(* Logix 5000 project; controller BigNumber Emulate 5570 rev 30.12; software revision 30.00 *)

TASK MainTask (periodic, rate 12000 ms, priority 1, watchdog 12000 ms) : MainProgram

MODULES
   Local : Emulate 5570 (ICP 3, rev 30.12)
       : vendor 1 type 0 code 15 (ICP 0, rev 1.1, Output RPI 50 ms)
END_MODULES

VAR_GLOBAL   (* controller tags *)
   SCAN_CYCLE_TIME : DINT; {access None}
END_VAR

PROGRAM MainProgram   (* main routine MainRoutine *)
VAR
   Add_c : DINT; {access None}
   Add_Digits : DINT; {access None}
   Add_i : DINT; {access None}
   Add_input_x : DINT[512]; {access None}
   Add_input_y : DINT[512]; {access None}
   Add_j : DINT; {access None}
   Add_Result : DINT[513]; {access None}
   Add_tmp : DINT;
   AddMul_2Base : DINT[250];
   AddMul_Base : DINT[249];
   AddMul_Digits : DINT;
   AddMul_exp_bitindx : DINT;
   AddMul_exp_blk : DINT;
   AddMul_i : DINT;
   AddMul_input_exp : DINT[249];
   AddMul_input_g : DINT[249];
   AddMul_j : DINT;
   AddMul_Result : DINT[500];
   Big_base : DINT; {access None}
   Big_Comp_i : DINT;
   Big_Comp_Res : DINT;
   Big_lb : DINT;
   Big_Ver : DINT;
   Div_Digits : DINT; {access None}
   Div_i : DINT; {access None}
   Div_input_x : DINT[500]; {access None}
   Div_input_y : DINT[500]; {access None}
   Div_j : DINT; {access None}
   Div_k : DINT; {access None}
   Div_m : DINT; {access None}
   Div_mul : DINT[500]; {access None}
   Div_q_Digits : DINT; {access None}
   Div_quotient : DINT[500]; {access None}
   Div_remainder : DINT[500]; {access None}
   Div_state : DINT; {access None}
   Div_sub_n : DINT; {access None}
   Div_x : DINT; {access None}
   Div_x_Digits : DINT; {access None}
   Div_y_Digits : DINT; {access None}
   Mul_c : DINT; {access None}
   Mul_Comp : DINT; {access None}
   Mul_Digits : DINT; {access None}
   Mul_i : DINT; {access None}
   Mul_input_x : DINT[513]; {access None}
   Mul_input_y : DINT[513]; {access None}
   Mul_j : DINT; {access None}
   Mul_q : DINT; {access None}
   Mul_Result : DINT[1025]; {access None}
   Mul_u : DINT; {access None}
   Mul_v : DINT; {access None}
   Mul_x : DINT; {access None}
   Mul_y : DINT; {access None}
   Sub_c : DINT; {access None}
   Sub_Digits : DINT; {access None}
   Sub_i : DINT; {access None}
   Sub_input_x : DINT[512]; {access None}
   Sub_input_y : DINT[512]; {access None}
   Sub_j : DINT; {access None}
   Sub_Result : DINT[512]; {access None}
END_VAR

ROUTINE BIGINTEGER_Add   (* structured text *)
   //Calculate the addition of big numbers.  Resource: page 594 of the handbook.
   //input positive big intergers  Add_input_x[] and Add_input_y[], each having UHF_sints base UHF_base digits.
   //output: the sum Add_Result[] in radix UHF_base representation.
   
   // Addition test
   (*if S:FS then
   	Add_Digits:= 10;  //the Digits of input.
   	UHF_base:= 10; //input in decimal
   	// Addition test
   	for Add_i:=0 to Add_Digits-1 by 1 do //assign value to input
   		Add_input_x[Add_i]:=9;
   		Add_input_y[Add_i]:=9;
   	end_for;
   end_if; *)
   
   //JSR(BIGINTEGER_Init);
   
   
   
   for Add_i:=0 to Add_Digits by 1 do
   	Add_Result[Add_i]:=0;  //Initialize the sum to 0.
   end_for;
   
   //Calculate the sum Add_input_x[] + Add_input_y[].
   Add_c.[0]:=0;   //Initialize carry to zero.
   
   for Add_j:=0 to Add_Digits-1 by 1 do
   	Add_Result[Add_j]:=Add_input_x[Add_j] + Add_input_y[Add_j] + Add_c; // Compute every digit of the sum.
   
   	Case Big_Ver OF
   	0:
   		if Add_Result[Add_j]> Big_base Then
   			Add_c:=1;
   		else
   			Add_c:=0;
   		End_if;
   		Add_Result[Add_j]:= Add_tmp mod Big_base;
   	1,2:
   		Add_c.[0]:=Add_Result[Add_j].[Big_lb];
   		Add_Result[Add_j].[Big_lb]:=0;	//最高位清零
   	End_Case;
   end_for;
   
   Add_Result[Add_Digits]:= Add_c;
   
   Add_c:=0;
   
END_ROUTINE

ROUTINE BIGINTEGER_AMul   (* structured text *)
   //Input: g ∈ G, whereGisanadditivegroup,andapositiveintegere = (e_t, e_t−1 ···e _1 e_ 0 ) 2 .
   //OUTPUT: e · g.
   
   
   //A←0.
   //2. For i from t down to 0 do the following:
   //2.1 A←A + A.
   //2.2 If e i = 1 then A←A + g.
   //3. Return(A).
   
   /////////////////////////////////////////////////////////////////////////////////////////////
   
   
   For AddMul_i:=0 to AddMul_Digits-1 by 1 Do
   	AddMul_Result[AddMul_i]:=0;
   End_For;
   AddMul_exp_bitindx:=29; //indexing 30bits
   AddMul_exp_blk:=AddMul_Digits-2;
   
   
   For AddMul_i:=AddMul_Digits-2 to 0 by -1 Do
   	While AddMul_exp_bitindx>=0 Do
   		if AddMul_i<> AddMul_Digits-2 or AddMul_exp_bitindx <> 29 Then
   			Add_Digits:= AddMul_Digits-1;
   				for Add_i:=0 to Add_Digits-1 by 1 do //assign value to input
   					Add_input_x[Add_i]:=AddMul_Result[Add_i];
   					Add_input_y[Add_i]:=AddMul_Result[Add_i];
   				end_for;
   			JSR(BIGINTEGER_Add);
   			for Add_i:=0 to Add_Digits by 1 do //
   				AddMul_Result[Add_i]:=Add_Result[Add_i];
   			end_for;
   
   			JSR(BIGINTEGER_Comparison);
   			If Big_Comp_Res=1 Then           //mod m
   				Sub_Digits:= AddMul_Digits-1;
   				for Sub_i:=0 to Sub_Digits-1 by 1 do //assign value to input
   					Add_input_x[Sub_i]:=AddMul_Result[Sub_i];
   					Add_input_y[Sub_i]:=AddMul_Base[Sub_i];
   				end_for;
   				JSR(BIGINTEGER_Sub);
   				for Sub_i:=0 to Add_Digits by 1 do //
   					AddMul_Result[Sub_i]:=Add_Result[Sub_i];
   				end_for;
   			End_If;
   
   		End_IF;
   
   
   
   		If AddMul_input_exp[AddMul_exp_blk].[AddMul_exp_bitindx] Then
   			Add_Digits:= AddMul_Digits-1;
   				for Add_i:=0 to Add_Digits-1 by 1 do //assign value to input
   					Add_input_x[Add_i]:=AddMul_Result[Add_i];
   					Add_input_y[Add_i]:=AddMul_input_g[Add_i];
   				end_for;
   			JSR(BIGINTEGER_Add);
   			for Add_i:=0 to Add_Digits by 1 do //
   				AddMul_Result[Add_i]:=Add_Result[Add_i];
   			end_for;
   
   			JSR(BIGINTEGER_Comparison);
   			If Big_Comp_Res=1 Then           //mod m
   				Sub_Digits:= AddMul_Digits-1;
   				for Sub_i:=0 to Sub_Digits-1 by 1 do //assign value to input
   					Add_input_x[Sub_i]:=AddMul_Result[Sub_i];
   					Add_input_y[Sub_i]:=AddMul_Base[Sub_i];
   				end_for;
   				JSR(BIGINTEGER_Sub);
   				for Sub_i:=0 to Add_Digits by 1 do //
   					AddMul_Result[Sub_i]:=Add_Result[Sub_i];
   				end_for;
   			End_If;
   
   		End_If;
   		AddMul_exp_bitindx:=AddMul_exp_bitindx-1;
   
   	End_while;
   
   
   	AddMul_exp_blk:=AddMul_exp_blk-1;
   	AddMul_exp_bitindx:=29;
   
   
   End_For;
   
   
   
   
   
END_ROUTINE

ROUTINE BIGINTEGER_Comparison   (* structured text *)
   Big_Comp_Res:=0;    //0: x>=y,  1: x<y
   
   
   Big_Comp_i:=AddMul_Digits-1;
   
   
   While Big_Comp_i>= 0 do
   
   	if AddMul_2Base[Big_Comp_i]< AddMul_Result[Big_Comp_i] Then
   	 	Big_Comp_Res:=1;
   		exit;
   	End_If;
   
   	Big_Comp_i:=Big_Comp_i-1;
   
   End_while;
   
   
   
END_ROUTINE

ROUTINE BIGINTEGER_Div   (* structured text *)
   //Calculate the division of big numbers.  Resource: page 598 of the handbook.
   //input positive big intergers  Div_input_x[] and Div_input_y[], Div_input_x[] having UHF_sints base UHF_base digits.
   //output: the quotient Div_quo[] and remainder Div_rem[] in radix UHF_base representation.
   
   (*if S:FS then
   	// division test
   	Div_state:=0;
    	Div_Digits:= 10;  //the Digits of input.
   	UHF_base:= 10; //input in decimal
   	for Div_i:=0 to Div_Digits-1 by 1 do   //assign value to input
   		Div_input_x[Div_i]:=9;
   	end_for;
   	for Div_i:=0 to (Div_Digits-1)/2 by 1 do
   		Div_input_y[Div_i]:=9;
   	end_for;
   end_if;*)
   
   	for Div_i:=Div_Digits-1 to 0 by -1 do  //Calculate the numbers of digit of Div_input_x[].
   		if Div_input_x[Div_i] <> 0 then
   			Div_x_Digits:= Div_i;
   			exit;
   		end_if;
   	end_for;
   
   	for Div_i:=Div_Digits-1 to 0 by -1 do  ////Calculate the numbers of digits of Div_input_y[].
   		if Div_input_y[Div_i] <> 0 then
   			Div_y_Digits:= Div_i;
   			exit;
   		end_if;
   	end_for;
   
   	Div_q_Digits:= Div_x_Digits - Div_y_Digits; //the numbers of digit of Div_quotient[].
   	for Div_i:=0 to Div_q_Digits by 1 do
   		Div_quotient[Div_i]:= 0;    //Initialize Div_quotient[] is zero.
   	end_for;
   
   	for Div_i:=0 to Div_x_Digits by 1 do
   		Div_mul[Div_i]:=0;
   	end_for;
   
   
   //When the dividend is less than the divisor, e.g Div_input_x is less than Div_input_y
   for Div_i:=Div_Digits-1 to 0 by -1 do
   	if Div_x_Digits <= Div_y_Digits and Div_input_x[Div_i] < Div_input_y[Div_i] then
   		Div_quotient[0]:=0;
   		for Div_i:=0 to Div_x_Digits by 1 do
   			Div_remainder[Div_i]:=Div_input_x[Div_i];
   		end_for;
   		exit;
   	else
   		Div_state:=1;
   	end_if;
   end_for;
   
   //When the dividend is equal to the divisor
   if Div_state=1 then
   	for Div_i:=Div_Digits-1 to 0 by -1 do
   		if Div_x_Digits = Div_y_Digits and Div_input_x[Div_i] = Div_input_y[Div_i] then
   			Div_quotient[0]:= 1;
   			Div_remainder[0]:= 0;
   		else
   			Div_state:=2;
   		end_if;
   	end_for;
   end_if;
   
   //When the dividend Div_input_x[] is greater than the divisor
   if Div_state=2 then
   	//Compute highest digit value of quotient Div_quotient[].
   	for Div_i:= Div_x_Digits to Div_q_Digits by -1 do  //compute Div_input_y[]*(power(UHF_base,(Div_q_Digits)).
   		Div_mul[Div_i]:= Div_input_y[Div_i-Div_q_Digits];
   	end_for;
   	for Div_i:= 0 to Div_q_Digits-1 by 1 do
   		Div_mul[Div_i]:= 0;
   	end_for;
   	for Div_i:=Div_x_Digits to 0 by -1 do  //Calculate the numbers of digit of Div_mul[]
   		if Div_mul[Div_i]<>0 then
   			Div_m:= Div_i;
   			exit;
   		end_if;
   	end_for;
   
   // Determine whether Div_input_x is greater than or equal to Div_input_y[]*(power(UHF_base,(Div_q_Digits)).
   	while Div_input_x[Div_x_Digits] >= Div_mul[Div_x_Digits] do
   
   		Div_quotient[Div_q_Digits]:=Div_quotient[Div_q_Digits] + 1;
   		Sub_Digits:=Div_x_Digits + 1;
   		for Div_k:=0 to Div_x_Digits by 1 do  //compute Div_input_x[]:=Div_input_x[]-Div_input_y[]*(power(UHF_base,(Div_q_Digits)).
   			Sub_input_x[Div_k]:= Div_input_x[Div_k];
   			Sub_input_y[Div_k]:= Div_mul[Div_k];
   		end_for;
   		JSR(BIGINTEGER_Sub);
   
   		for Div_k:= 0 to Div_x_Digits by 1 do  //Updated Div_input_x[] after subtraction.
   			Div_input_x[Div_k]:= Sub_Result[Div_k];
   		end_for;
   
   	end_while;
   
   	for Div_i:=0 to Div_x_Digits by 1 do   //cleared before the next time call
   		Div_mul[Div_i]:= 0;
   	end_for;
   //----------------------------------------------------------------------------------
   	//compute other digit value of quotient Div_quotient[].
   	for Div_j:= Div_x_Digits to Div_y_Digits+1 by -1 do
   
   		if Div_input_x[Div_j]= Div_input_y[Div_y_Digits] then
   			Div_quotient[Div_j-Div_y_Digits-1]:= Big_base-1;
   		else
   			Div_quotient[Div_j-Div_y_Digits-1]:= (Div_input_x[Div_j] * Big_base + Div_input_x[Div_j-1]) / Div_input_y[Div_y_Digits];
   		end_if;
   
   		while (Div_quotient[Div_j-Div_y_Digits-1]*(Div_input_y[Div_y_Digits]*Big_base+Div_input_y[Div_y_Digits-1])) >
   			(Div_input_x[Div_j]*Big_base*Big_base+Div_input_x[Div_j-1]*Big_base+Div_input_x[Div_j-2]) do
   				Div_quotient[Div_j-Div_y_Digits-1]:= Div_quotient[Div_j-Div_y_Digits-1] - 1;
   		end_while;
   
   		//compute Div_quotient[Div_j-Div_y_sints-1]*Div_input_y[]*(power(UHF_base,(Div_j-Div_y_sints-1))
   		for Div_k:= Div_j to Div_j-Div_y_Digits-1 by -1 do
   			Div_mul[Div_k]:= Div_input_y[Div_k-(Div_j-Div_y_Digits-1)];  //compute Div_input_y[]*(power(UHF_base,(Div_j-Div_y_sints-1)).
   		end_for;
   		for Div_k:=0 to Div_j-Div_y_Digits-2 by 1 do
   			Div_mul[Div_k]:=0;
   		end_for;
   
   		Mul_Digits:=Div_x_Digits + 1;
   		for Div_k:=0 to Div_x_Digits by 1 do
   			Mul_input_y[Div_k]:= Div_mul[Div_k];  //assign value of Div_mul[] to Mul_input_y[]
   		end_for;
   		//	Mul_input_x[0]:= Div_quotient[Div_j-DIV_y_Digits-1];  //assign value of Div_quo[Div_j-Div_y_sints-1] to Mul_input_x[].
   		Mul_input_x[0]:= Div_quotient[Div_j-Div_y_Digits-1];
   		for Div_k:=1 to Mul_Digits-1  by 1 do
   			Mul_input_x[Div_k]:= 0;  //assign value of Div_mul[] to Mul_input_y[]
   		end_for;
   		JSR(BIGINTEGER_Mul);
   
   		//compute Div_input_x[]-Div_quo[Div_j-Div_y_sints-1]*Div_input_y[]*(power(UHF_base,(Div_j-Div_y_sints-1)).
   		Sub_Digits:=Div_x_Digits + 1;
   		for Div_k:=0 to Div_x_Digits by 1 do
   			Sub_input_y[Div_k]:= Mul_Result[Div_k]; //assign value of Mul_Result[] to Sub_input_y[]
   		end_for;
   		for Div_k:=0 to Div_x_Digits by 1 do
   			Sub_input_x[Div_k]:= Div_input_x[Div_k];  //assign value of Div_input_x[] to Sub_input_x[]
   		end_for;
   		JSR(BIGINTEGER_Sub);
   
   		for Div_k:=Div_x_Digits to 0 by -1 do
   			if Sub_Result[Div_k] <> 0 then
   				Div_sub_n:= Div_k;
   				exit;
   			end_if;
   		end_for;
   
   		for Div_k:=0 to Div_x_Digits by 1 do
   	 		Div_input_x[Div_k]:= Sub_Result[Div_k];  //print the remainder.
   		end_for;
   
   		if Div_input_x[Div_sub_n] < 0 then  //compute Div_input_x[]:= Div_input_x[]+Div_input_y[]*(power(UHF_base,(Div_j-Div_y_sints-1)).
   			Add_Digits:=Div_x_Digits + 1;
   			for Div_i:=0 to Div_x_Digits by 1 do
   				Add_input_x[Div_i]:= Sub_Result[Div_i];
   			end_for;
   			for Div_i:=0 to Div_x_Digits by 1 do
   				Add_input_y[Div_i]:= Div_mul[Div_i];
   			end_for;
   			JSR(BIGINTEGER_Add);
   			Div_quotient[Div_j-Div_y_Digits-1]:=Div_quotient[Div_j-Div_y_Digits-1]-1;
   
   			for Div_k:=0 to Div_x_Digits by 1 do
   				Div_input_x[Div_k]:= Add_Result[Div_k];  //print the remainder.
   			end_for;
   		end_if;
   	end_for;
   
   	for Div_i:=0 to Div_y_Digits by 1 do
   		Div_remainder[Div_i]:=Div_input_x[Div_i];
   	end_for;
   end_if;
   
   for Div_i:=0 to Div_Digits-1 by 1 do
   	Div_input_x[Div_i]:=0;
   	Div_input_y[Div_i]:=0;
   end_for;
   
   
END_ROUTINE

ROUTINE BIGINTEGER_Init   (* structured text *)
   Case Big_Ver Of
   0:
   	Big_lb := 4;      // base =10
   	Big_base:=10;
   
   1:
   
   	Big_lb := 15;    // for  both mul/div and add/sub, b=2^15
   	Big_base:=32768;
   
   2:
   	Big_lb := 30;   //for addition only        b=2^30
   	Big_base:=0;
   	Big_base.[30]:=1;
   	AddMul_Digits:=9; //for AddMul
   End_Case;
END_ROUTINE

ROUTINE BIGINTEGER_Mul   (* structured text *)
   //Calculate the multiplication of big numbers.  Resource: page 595 of the handbook.
   //input: positive big intergers  Mul_input_x[] and Mul_input_y[], each having UHF_sints base UHF_base digits.
   //output: the result Mul_Result[] in radix UHF_base representation with 2*(UHF_sints-1) digits.
   
   
   // multiplication test
   (*if S:FS then
   	Mul_Digits:= 512;  //the Digits of input.
   	UHF_base:= 10; //input in decimal
   	Mul_v:=0;
   	Mul_compute:=0;
   	Mul_u:=0;
   	UHF_c:=0;
   	for Mul_i:=0 to Mul_Digits-1 by 1 do   //assign value to input
   		Mul_input_x[Mul_i]:=9;
   		Mul_input_y[Mul_i]:=9;
   	end_for;
   end_if;*)
   
   
   	for Mul_i:=0 to 2*Mul_Digits-1 by 1 do
   		Mul_Result[Mul_i]:=0;  //Initialize the result of multiplication to 0.
   	end_for;
   
   	for Mul_i:=0 to Mul_Digits-1 by 1 do
   		Mul_c:=0;
   		for Mul_j:=0 to Mul_Digits by 1 do
   			Mul_Comp:= Mul_Result[Mul_i+Mul_j]+(Mul_input_y[Mul_j]*Mul_input_x[Mul_i]+Mul_c); //compute the result of every digit of Mul_input_y multiply one digit of Mul_input_x.
   	//UHF_Mul_input_x[UHF_i]*UHF_Mul_input_y[UHF_j] = (UHF_Mul_u||UHF_Mul_v)UHF_base.
   			if Mul_Comp > Big_base-1 then  //if the Mul_compute is greater than UHF_base-1, then split Mul_compute.
   				Mul_v:= Mul_Comp mod Big_base;
   				Mul_u:= Mul_Comp / Big_base;
   			else
   				Mul_v:= Mul_Comp;
   				Mul_u:=0;
   			end_if;
   			Mul_Result[Mul_i+Mul_j]:=Mul_v; //Result of multiplication
   			Mul_c:= Mul_u;   //the carry is equal to left half bits of Mul_compute.
   		end_for;
   	end_for;
   
   	for Mul_i:=0 to Mul_Digits-1 by 1 do
   		Mul_input_x[Mul_i]:=0;
   		Mul_input_y[Mul_i]:=0;
   	end_for;
   
   	Mul_u:=0;
   	Mul_v:=0;
   
   
   
   
   
END_ROUTINE

ROUTINE BIGINTEGER_Sub   (* structured text *)
   //Calculate the  subtraction of big numbers.  Resource: page 595 of the handbook.
   //input positive big intergers  Sub_input_x[] and Sub_input_y[], each having UHF_sints base UHF_base digits with x > y.
   //output: the result Sub_Result[] in radix UHF_base representation.
   
   // Subtraction test
   (*if S:FS then
   	Sub_Digits:= 10;  //the Digits of input.
   	UHF_base:= 10; //input in decimal
   	for Sub_i:=0 to Sub_Digits-1 by 1 do  //assign value to input
   		Sub_input_x[Sub_i]:=9;
   		Sub_input_y[Sub_i]:=6;
   	end_for;
   end_if;*)
   
   
   //JSR(BIGINTEGER_Init);
   
   
   for Sub_i:=0 to Sub_Digits-1 by 1 do
   	Sub_Result[Sub_i]:=0;  //Initialize the sum to 0.
   end_for;
   
   //Calculate the result Sub_input_x[] - Sub_input_y[].
   Sub_c:=0;   //Initialize carry to zero.
   
   for Sub_j:=0 to Sub_Digits-1 by 1 do
   
   	Sub_Result[Sub_j]:= Sub_input_x[Sub_j]-Sub_input_y[Sub_j]-Sub_c;
   	Add_c.[0]:=Add_Result[Add_j].[Big_lb];
   	Case Big_Ver OF
   		0:
   			Add_Result[Sub_j]:= Add_tmp MOD Big_base;
   		1:
   			Add_Result[Sub_j]:= Add_Result[Sub_j] AND 16#7FFF;
   		2:
   			//Add_Result[Sub_j]:= Add_Result[Sub_j] AND 16#3FFFFFFF‬;
   			Add_Result[Sub_j].[30]:=0;
   			Add_Result[Sub_j].[31]:=0;
   
   	End_Case;
   
   	  // Compute every digit of the subtraction.
   end_for;
   
   Add_c:=0;
   
END_ROUTINE

ROUTINE BIGINTEGER_Test   (* structured text *)
   (*Big_Ver:=2;
   
   Add_Digits:=2;
   Add_input_x[0]:=-1;
   
   Add_input_x[1]:=12345;
   
   Add_input_y[0]:=-3;
   
   Add_input_y[1] := -29747;
   
   
   JSR(BigNumber_Add);  *)
   
   Big_Ver:=2;
   
   JSR(BIGINTEGER_Init);
   
   if S:FS then
   //addmul test
   	for AddMul_i:=0 to AddMul_Digits-2 by 1 do
   		AddMul_Base[AddMul_i]:=-1 AND 16#3FFFFFFF;
   		AddMul_input_g[AddMul_i]:=5678;
   		AddMul_input_exp[AddMul_i]:=-1 AND 16#3FFFFFFF;
   	end_for;
   	Mul_Digits:=AddMul_Digits-2;
   	Mul_input_y[Mul_i]:=2;
   	for Mul_i:=0 to Mul_Digits-1 by 1 do   //assign value to input
   		Mul_input_x[Mul_i]:=AddMul_Base[Mul_i];
   		if Mul_i=0 Then
   			Mul_input_y[Mul_i]:=2;
   		else
   			Mul_input_y[Mul_i]:=0;
   		End_If;
   	end_for;
   	JSR(BIGINTEGER_Mul);
   
   	for Mul_i:=0 to Mul_Digits by 1 do
   		AddMul_2Base[Mul_i]:=Mul_Result[Mul_i];
   	end_for;
   
   
   end_if;
   
   JSR(BIGINTEGER_AMul);
   
END_ROUTINE

ROUTINE MainRoutine   (* ladder *)
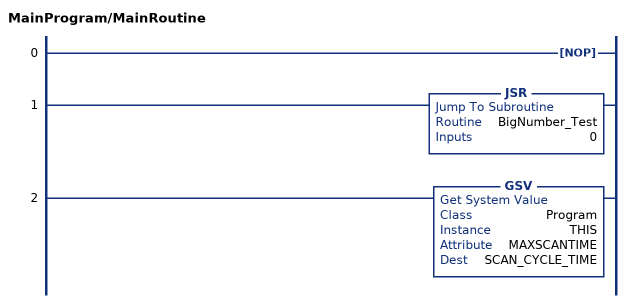
   0: NOP();
   1: JSR(BigNumber_Test,0);
   2: GSV(Program,THIS,MAXSCANTIME,SCAN_CYCLE_TIME);
END_ROUTINE
END_PROGRAM
